{attribute addProperty BoxType "EK1100-0000-0018"}
{attribute addProperty Id "Beckhoff_EJ5xxxEK1122Beckhoff_EJ5xxxEK1122_0744EC7C162A_0001_EJ5002_0000_0016EJ5002_8228306817822.25A_0002_EJ5002_0000_0017EJ5002_960CC6F117822.25A_0003_EJ5101_0000_0016EJ5101_6012872616220.25A_0004_EJ5151_0000_0016EJ5151_0AC1A36D19424.25"}
{attribute addProperty CRC "3743602083"}
{attribute addProperty SizeInBites "728"}
{attribute addProperty SizeInBytes "91"}
TYPE Beckhoff_EJ5xxx_DF22D5A3 EXTENDS EK1100_179A0949 :
STRUCT
	{attribute addProperty Name "Beckhoff_EJ5xxxEK1122"}
	Beckhoff_EJ5xxxEK1122 : Beckhoff_EJ5xxxEK1122_0744EC7C;
	{attribute addProperty Name "A_0001_EJ5002_0000_0016"}
	A_0001_EJ5002_0000_0016 : EJ5002_82283068;
	{attribute addProperty Name "A_0002_EJ5002_0000_0017"}
	A_0002_EJ5002_0000_0017 : EJ5002_960CC6F1;
	{attribute addProperty Name "A_0003_EJ5101_0000_0016"}
	A_0003_EJ5101_0000_0016 : EJ5101_60128726;
	{attribute addProperty Name "A_0004_EJ5151_0000_0016"}
	A_0004_EJ5151_0000_0016 : EJ5151_0AC1A36D;
END_STRUCT
END_TYPE

(* stored: Version 1.2.0.0, ProductVersion 3.1.4024.9
   DUT Beckhoff_EJ5xxx_DF22D5A3: Id {f54fdc01-3451-4105-a4ab-adb30e2fff57} *)
